(* IEC 61131-3 sources: stc/tests/fixtures/valid_ast, 5 files *)

(* ---- simple_type_alias.st ---- *)
(* Copyright (C) 2021-2026 Manuele Conti
   SPDX-License-Identifier: GPL-2.0-or-later
   Summary: Exercises parsing of a derived elementary type alias. *)

TYPE
    MyInt : INT;
    MyBool : BOOL;
END_TYPE

(* ---- case_and_for.st ---- *)
(* Copyright (C) 2021-2026 Manuele Conti
   SPDX-License-Identifier: GPL-2.0-or-later
   Summary: Exercises CASE selection and FOR iteration AST nodes. *)

FUNCTION normalize_mode : INT
VAR_INPUT
    mode_value: INT;
END_VAR
VAR
    index_value: INT;
END_VAR
    CASE mode_value OF
        0: normalize_mode := 10;
        1, 2: normalize_mode := 20;
    ELSE
        normalize_mode := 0;
    END_CASE;
    FOR index_value := 0 TO 3 BY 1 DO
        normalize_mode := normalize_mode + index_value;
    END_FOR;
END_FUNCTION

(* ---- direct_variables.st ---- *)
(* Copyright (C) 2021-2026 Manuele Conti
   SPDX-License-Identifier: GPL-2.0-or-later
   Summary: Exercises parsing of directly represented IEC variables. *)

FUNCTION read_input_word : INT
VAR_INPUT
    fallback_value: INT;
END_VAR
    read_input_word := %IW0;
END_FUNCTION

(* ---- function_block_counter.st ---- *)
(* Copyright (C) 2021-2026 Manuele Conti
   SPDX-License-Identifier: GPL-2.0-or-later
   Summary: Exercises a stateful counter function-block declaration. *)

FUNCTION_BLOCK Counter
VAR_INPUT
    reset_value : BOOL;
END_VAR
VAR_OUTPUT
    count_value : INT;
END_VAR
    IF reset_value THEN
        count_value := 0;
    ELSE
        count_value := count_value + 1;
    END_IF;
END_FUNCTION_BLOCK

(* ---- expanded_grammar.st ---- *)
(* Copyright (C) 2021-2026 Manuele Conti
   SPDX-License-Identifier: GPL-2.0-or-later
   Summary: Covers declarations, literals, calls, programs, and control flow. *)

TYPE
    SampleArray : ARRAY [0..3] OF INT;
    SampleStruct : STRUCT
        count_value : INT;
        label_text : STRING[16];
    END_STRUCT;
END_TYPE

FUNCTION normalize_sample : INT
VAR_INPUT
    raw_value: INT;
END_VAR
VAR
    values: ARRAY [0..3] OF INT := [1, 2, 3, 4];
    status_text: STRING[16] := 'running';
    created_on: DATE := D#2026-07-17;
    started_at: TIME_OF_DAY := TOD#12:34:56.7;
    sample_stamp: DATE_AND_TIME := DT#2026-07-17-12:34:56.7;
    timeout_value: TIME := T#1H;
END_VAR
    CASE raw_value OF
        0: normalize_sample := MIN(IN1 := raw_value, IN2 := 10);
        1, 2: normalize_sample := LIMIT(MN := 0, IN := raw_value, MX := 10);
    ELSE
        normalize_sample := MAX(IN1 := raw_value, IN2 := 0);
    END_CASE;

    FOR raw_value := 0 TO 3 BY 1 DO
        normalize_sample := normalize_sample + values[raw_value];
    END_FOR;
END_FUNCTION

PROGRAM SampleProgram
VAR
    current_value: INT;
END_VAR
    current_value := normalize_sample(raw_value := current_value);
END_PROGRAM
